FUNCTION_BLOCK Insertion //2d insertion that combines a slider (alignment) and screw (push)
VAR_INPUT //interface references to existing drives
	slider : I_EncodedDrive;
	screw : I_ContinuousDrive;
END_VAR
VAR_OUTPUT
	contact AT %I* : BOOL;
	
	active : BOOL;
	error : BOOL;
	home : BOOL;
	
	homingComplete : BOOL;
	
	sliderPos : LREAL;
END_VAR
(*
VAR
	slider : LinearDrive_Encoded; //I_PositionalDrive;
	screw : LinearDrive_Continuous; //I_ContinuousDrive;
END_VAR
*)
(*
this FB encapsulates 2 linear drives into a generic insertion machine
both drives should be declared externally in Hardware GVL as a concrete FB
Insertion instance should be declared and called in module scope, with the drives from Hardware GVL passed in by Interface reference
*)

homingComplete := slider.HomeSet AND screw.HomeSet;

active := slider.Active OR screw.Active;
error := slider.Error OR screw.Error;
home := slider.AtHome AND screw.AtHome;

sliderPos := slider.CurrentPosition;

METHOD align : BOOL
VAR_INPUT
	targetPos : REAL;
END_VAR
slider.moveAbsolute(newTarget := targetPos);
END_METHOD

METHOD homingSequence : BOOL
VAR_INPUT
END_VAR
IF NOT slider.homeSet THEN
	slider.homingSequence();
END_IF

IF NOT screw.homeSet THEN
	screw.homingSequence();
END_IF

homingSequence := homingComplete;
END_METHOD

METHOD press : BOOL
VAR_INPUT
END_VAR
IF NOT contact THEN
	screw.moveContinuous(newDirection := MC_Negative_Direction);
END_IF
END_METHOD

METHOD release : BOOL
VAR_INPUT
END_VAR
screw.moveContinuous(newDirection := MC_Positive_Direction);
END_METHOD

METHOD reset : BOOL
VAR_INPUT
END_VAR
slider.reset();
screw.reset();
END_METHOD

METHOD stop : BOOL
VAR_INPUT
END_VAR
screw.stop();
slider.stop();
END_METHOD

METHOD toHome : BOOL
VAR_INPUT
END_VAR
slider.toHome();
screw.toHome();

toHome := slider.AtHome AND screw.AtHome;
END_METHOD

END_FUNCTION_BLOCK

(* stored: Version 1.1.0.1, ProductVersion 3.1.4024.11
   POU Insertion: Id {502e06bc-53e2-4b1f-90c3-fdcb2d93fff1}, SpecialFunc None
   Method align: Id {64e46e12-9cfc-4e03-9108-28988a144d43}
   Method homingSequence: Id {7c5357a6-8a67-4a9c-9b11-a9929607beee}
   Method press: Id {e55c5f15-8abc-4542-a690-5e6367be3b31}
   Method release: Id {33c0891b-5c36-438e-984e-bc3daf298105}
   Method reset: Id {21971230-04b8-4583-b08d-9d3fcf007286}
   Method stop: Id {d0ed2cc3-be18-4ec0-a385-1359d2d26244}
   Method toHome: Id {8609ef5e-d448-4bc3-a23e-98291f314b18} *)
